{attribute 'object_name' := 'sta_WaitPaperGone'}
METHOD PROTECTED sta_WaitPaperGone : BOOL
// state implemetation
//--------------------------------------------------------------------------------------
// Entry action
	IF (me.StateMachine.intState<>me.StateMachine.intStateLastCycle) THEN
		me.StateMachine.intStateLastCycle := me.StateMachine.intState;

		IF (SIf.Cfg.bolRaxEnable) THEN
			p_fbRAX^.CtrlCIf^.Job.intACmd := cCMD_STOP;
		ELSE
			IF (SIf.Cur.rInOutPosition.uinInput <> p_fbMalteser^.CtrlSIf^.Cur.uintActualPosition)
			  AND SIf.Cfg.bolPositionMalteserEnable THEN
				p_fbMalteser^.CtrlSIf^.Par.intTurnDirection := E_TURN_DIRECTION.AUTOMATIC;
				p_fbMalteser^.CtrlSIf^.Par.uinPositionToGo := SIf.Cur.rInOutPosition.uinInput;
				p_fbMalteser^.CtrlCIf^.Job.intACmd := MDC_CmdState.cCMD_PREPOSITION;
			END_IF
		END_IF
		
		me.SubStateMachine.intState := cSTA_WaitPaperGone;
		me.SubStateMachine.intStateNext := cSTA_WaitPaperGone;
	END_IF


//--------------------------------------------------------------------------------------
// Cyclic action
	IF (me.StateMachine.intState=me.StateMachine.intStateLastCycle) THEN
		// sub state machine for sequence
		CASE me.SubStateMachine.intState OF
			//--------------------------------------------------------------------------------------
			PTS_CmdState.cSTA_WaitPaperGone:
				IF NOT SIf.In.bolPaperAvailable.intern THEN
					me.SubStateMachine.intStateNext := cSUB_DELAYbusy;
				END_IF

				IF (me.SubStateMachine.udiTimeInState_ms > SIf.Par.udiPaperBarcodeToInputSensorTime) THEN
					pfbAlarmCtrl^.setAlarm(CIf.Info.intCtrlId,INT_TO_UINT(E_ALM_PTS.PaperTransport),0,ADR(SIf.Alm),E_AlmState.RST,CIf.Job.eMe_ActivAlmClass);
					me.StateMachine.intStateNext := BASE_PLC.cSTA_ERROR;
				END_IF
			//--------------------------------------------------------------------------------------
			PTS_CmdState.cSUB_DELAYbusy:
			  	IF SIf.Par.udiPaperOutTurnDelayTime = 0 THEN
					me.StateMachine.intStateNext := PTS_CmdState.cSTA_TurnEmptyBusy;
				ELSE	
					IF (me.StateMachine.udiTimeInState_ms > SIf.Par.udiPaperOutTurnDelayTime) THEN
						me.StateMachine.intStateNext := PTS_CmdState.cSTA_TurnEmptyBusy;
					END_IF
				END_IF
			//--------------------------------------------------------------------------------------
			PTS_CmdState.cSUB_PREPOSITIONbusy:
				IF (SIf.Cfg.bolRaxEnable = FALSE) THEN
					IF (p_fbMalteser^.CtrlCIf^.Job.intState = MDC_CmdState.cSTA_PREPOSITION) THEN
						p_fbMalteser^.CtrlCIf^.Job.intACmd := BASE_PLC.cCMD_RUN;
						me.SubStateMachine.intStateNext := PTS_CmdState.cSUB_WAIT_DONE;
					END_IF
				END_IF
			//--------------------------------------------------------------------------------------
			PTS_CmdState.cSUB_WAIT_DONE:
				IF (p_fbMalteser^.CtrlCIf^.Job.intState = MDC_CmdState.cSTA_InPosition) THEN
					me.SubStateMachine.intStateNext := cSTA_WaitPaperGone;
				END_IF
		END_CASE
	END_IF


//--------------------------------------------------------------------------------------
// Exit action
	IF (me.StateMachine.intState<>me.StateMachine.intStateNext) THEN
		;
	END_IF
END_METHOD

{attribute 'object_name' := 'StateMachine'}
METHOD PROTECTED StateMachine : BOOL
SUPER^.StateMachine();

// main statemachine of base controller
CASE me.StateMachine.intState OF
    PTS_CmdState.cSTA_STANDBYBusy: 
        THIS^.sta_STANDBYBusy();
    PTS_CmdState.cSTA_STANDBY: 
        THIS^.sta_STANDBY();
    BASE_PLC.cSTA_RUNBusy: 
        THIS^.sta_RUNBusy();
    BASE_PLC.cSTA_RUN: 
        THIS^.sta_RUN();
    BASE_PLC.cSTA_STOPBusy: 
        THIS^.sta_STOPBusy();
    BASE_PLC.cSTA_STOP: 
        THIS^.sta_STOP();
    PTS_CmdState.cSTA_PaperDelayBusy: 
        THIS^.sta_PaperDelayBusy();
    PTS_CmdState.cSTA_TurnPaperBusy: 
        THIS^.sta_TurnPaperBusy();
    PTS_CmdState.cSTA_WaitPaperGone: 
        THIS^.sta_WaitPaperGone();
    PTS_CmdState.cSTA_TurnEmptyBusy: 
        THIS^.sta_TurnEmptyBusy();
    PTS_CmdState.cSTA_InitializeBusy: 
        THIS^.sta_InitializeBusy();
    PTS_CmdState.cSTA_WaitPaper: 
        THIS^.sta_WaitPaper();
    PTS_CmdState.cSTA_GetItemBusy: 
        THIS^.sta_GetItemBusy();
END_CASE;
END_METHOD

END_FUNCTION_BLOCK

// POUs/Controller/Utility/Data Channel/OvenMessage/FB_OvenSendDch
FUNCTION_BLOCK FB_OvenSendDch EXTENDS FB_DataChannelSendBase IMPLEMENTS I_DataChannelSend
VAR
	/// Saber Inteface Variables
	/// -----------------------------------------------------------------
	m_pOutputData: POINTER TO T_Oven_DCH;
END_VAR

SUPER^();

{attribute 'object_name' := 'InitChannel'}
METHOD InitChannel : BOOL
VAR_INPUT
	udiDataSize: UDINT;
	pOutputData: POINTER TO BYTE;
END_VAR
InitChannel := FALSE;

IF udiDataSize > 0 THEN
	IF pOutputData <> TC3_MEMMAN.NULL THEN
		m_uinDataSize := udiDataSize;
		m_pOutputData := pOutputData;
		m_eState := E_PlcSaberDHCState.Init;
		InitChannel := TRUE;
	END_IF
END_IF
END_METHOD

{attribute 'object_name' := 'SendData'}
METHOD SendData : BOOL
VAR_INPUT
	udiDataSize: UDINT;
	pData: POINTER TO BYTE;
END_VAR
SendData := FALSE;

IF m_eState = E_PlcSaberDHCState.WaitForJob THEN
	IF (udiDataSize > 0 ) AND (pData <> TC3_MEMMAN.NULL) THEN
		TC2_SYSTEM.MEMCPY(destAddr := m_pOutputData, srcAddr := pData, n := udiDataSize);
		m_eState := E_PlcSaberDHCState.SendData;	
		SendData := TRUE;
	END_IF	
END_IF
END_METHOD

END_FUNCTION_BLOCK
